// TIA Portal V15.1 export
// export: Created 2022-12-20T09:13:23.330167Z, ExportSetting None, DisplayName Totally Integrated Automation Portal, DisplayVersion V15.1 Update 1, DisplayName TIA Portal Openness, DisplayVersion V15.1, DisplayName SINAMICS Startdrive Advanced, DisplayVersion V15.1, DisplayName G130, G150, S120, S150, SINAMICS MV, S210, DisplayVersion V15.1, DisplayName G110M, G120, G120C, G120D, G120P, DisplayVersion V15.1, DisplayName STEP 7 Professional, DisplayVersion V15.1 Update 1, DisplayName STEP 7 Safety, DisplayVersion V15.1, DisplayName WinCC Professional, DisplayVersion V15.1 Update 1, DisplayName SIMATIC Visualization Architect, DisplayVersion V15.1
FUNCTION_BLOCK "SA01_FB"   // FB900, LAD
TITLE = SA01 FB
{ S7_Optimized_Access := 'FALSE' }
// The block is used to control the function blocks that are needed on SA01 level
// stored: AutoNumber false, CodeModifiedDate 2022-12-20T09:13:23.330167Z, SetENOAutomatically False
   VAR
      Mode : "Mode_SA_FB";   // Mode
   END_VAR
BEGIN

REGION Network 1: Call Mode FB
   // Depending on the inputs preconditions, commands, alarms, HMI and input from Safety Area (SA) Determine the current function, mode of operandi, and state.
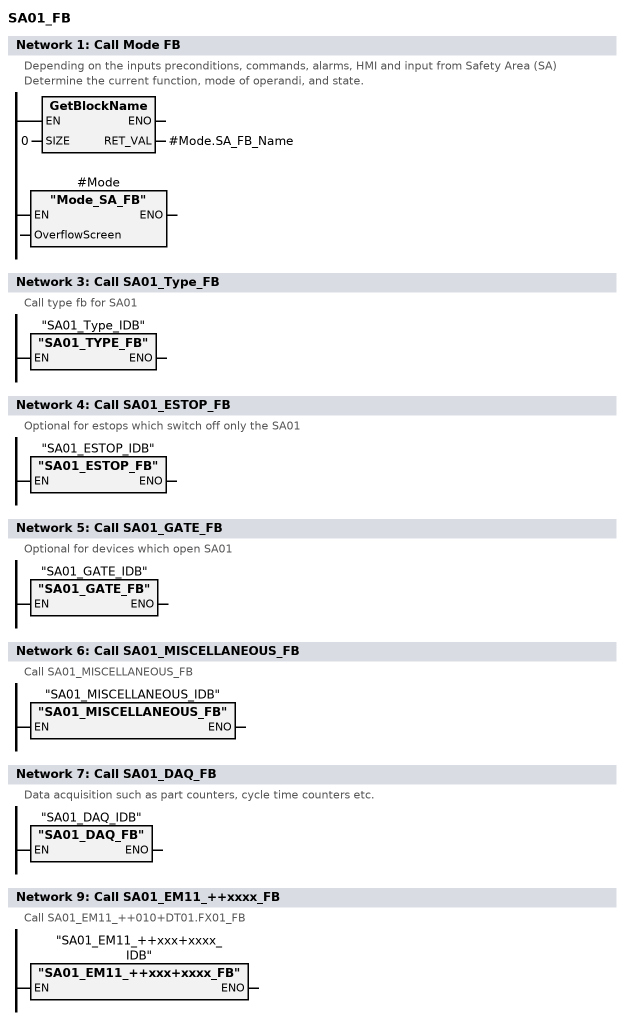
   RUNG wire#powerrail
      GetBlockName(size := 0, Ret_Val => #Mode.SA_FB_Name)
   END_RUNG
   RUNG wire#powerrail
      #Mode(OverflowScreen :=)
   END_RUNG
   // the same network as SCL:
   #Mode.SA_FB_Name := GetBlockName(size := 0);
   #Mode();   // "Mode_SA_FB"
END_REGION

REGION Network 2: ***SA01***
END_REGION

REGION Network 3: Call SA01_Type_FB
   // Call type fb for SA01
   RUNG wire#powerrail
      "SA01_Type_IDB"()
   END_RUNG
   // the same network as SCL:
   "SA01_Type_IDB"();   // "SA01_TYPE_FB"
END_REGION

REGION Network 4: Call SA01_ESTOP_FB
   // Optional for estops which switch off only the SA01
   RUNG wire#powerrail
      "SA01_ESTOP_IDB"()
   END_RUNG
   // the same network as SCL:
   "SA01_ESTOP_IDB"();   // "SA01_ESTOP_FB"
END_REGION

REGION Network 5: Call SA01_GATE_FB
   // Optional for devices which open SA01
   RUNG wire#powerrail
      "SA01_GATE_IDB"()
   END_RUNG
   // the same network as SCL:
   "SA01_GATE_IDB"();   // "SA01_GATE_FB"
END_REGION

REGION Network 6: Call SA01_MISCELLANEOUS_FB
   // Call SA01_MISCELLANEOUS_FB
   RUNG wire#powerrail
      "SA01_MISCELLANEOUS_IDB"()
   END_RUNG
   // the same network as SCL:
   "SA01_MISCELLANEOUS_IDB"();   // "SA01_MISCELLANEOUS_FB"
END_REGION

REGION Network 7: Call SA01_DAQ_FB
   // Data acquisition such as part counters, cycle time counters etc.
   RUNG wire#powerrail
      "SA01_DAQ_IDB"()
   END_RUNG
   // the same network as SCL:
   "SA01_DAQ_IDB"();   // "SA01_DAQ_FB"
END_REGION

REGION Network 8: ***ST 10***
END_REGION

REGION Network 9: Call SA01_EM11_++xxxx_FB
   // Call SA01_EM11_++010+DT01.FX01_FB
   RUNG wire#powerrail
      "SA01_EM11_++xxx+xxxx_IDB"()
   END_RUNG
   // the same network as SCL:
   "SA01_EM11_++xxx+xxxx_IDB"();   // "SA01_EM11_++xxx+xxxx_FB"
END_REGION
END_FUNCTION_BLOCK
